# EPICS substitutions: utcaApp/Db/fofb_cc.substitutions
file db/scan_task.template {
    {}
}

file db/fofb_cc.template {
    {}
}

file db/fofb_cc_channel.template {
    pattern {FOFB_CHAN, ADDR}
    {"CH0", "0"}
    {"CH1", "1"}
    {"CH2", "2"}
    {"CH3", "3"}
    {"CH4", "4"}
    {"CH5", "5"}
    {"CH6", "6"}
    {"CH7", "7"}
}
